{attribute 'linkalways'}
INTERFACE CommandStatus EXTENDS __SYSTEM.IQueryInterface

{attribute 'monitoring' := 'call'}
PROPERTY Busy : BOOL
GET
END_GET
END_PROPERTY

{attribute 'monitoring' := 'call'}
PROPERTY Done : BOOL
GET
END_GET
END_PROPERTY

{attribute 'monitoring' := 'call'}
PROPERTY Error : BOOL
GET
END_GET
END_PROPERTY

{attribute 'monitoring' := 'call'}
PROPERTY ErrorMessage : T_MaxString
GET
END_GET
END_PROPERTY

END_INTERFACE

(* stored: Version 1.1.0.1, ProductVersion 3.1.4024.15
   Itf CommandStatus: Id {640d2fb6-26ec-443c-a114-50dd19f0daa9}
   Property Busy: Id {4c2439e9-25fa-4a36-8fd0-4c79981cad60}
   Get Get: Id {ee70d7ab-49f3-463b-98f3-7386c1ba53c9}
   Property Done: Id {00363a4c-5a65-4f2b-ae4d-7cbe9769131d}
   Get Get: Id {ffd651f6-5507-4575-9c02-84fbbd175f1a}
   Property Error: Id {bfc3a5fe-2755-49d4-a606-8b367a1f3603}
   Get Get: Id {6b7e29ad-592c-4d26-a097-c6adae0f1094}
   Property ErrorMessage: Id {4eb8607d-b69d-43f1-a399-0771c18fef3d}
   Get Get: Id {63fe3413-d811-4454-8aa4-2d944fcf29c6} *)
